Staubli VAL3: Piramide.pgx

program Piramide()
  local num j
  local num k
  local num i
  local num l
begin
  //Mueve el brazo para crear una pirámide en 3D.

  // Se desplaza a la posicion de espera
  pEspera=appro(pPieza,{0,0,-50,0,0,0})
  movej(pEspera,tVentosa,mNomSpeed)
  waitEndMove()

  //Ciclo
  while !bTermina
    if bStartPiramide
      // Bucle de plantas
      for i = 0 to nPlantas - 1
        // Bucle de filas
        for j = 0 to nPlantas - nNivel - 1
          // Bucle de piezas para fila central y superiores
          for k = 0 to nPlantas - nNivel - nFila - 1
            // Se espera la orden de pieza preparada para continuar
            sMensaje="pulse 'enter' para continuar"
            wait(bPiezaPreparada)
            bPiezaPreparada=false
            sMensaje=""

            pObjetivo = appro(pCentro,{nX,(nLPieza/2)*(nPlantas-nNivel-nFila-1)-nY,-nZ,0,0,0})
            call pick(pPieza,tVentosa,mNomSpeed,mVelApprox)
            call place(pObjetivo,tVentosa,mNomSpeed,mVelApprox)
            nY=nY+nLPieza
          endFor
          // Nueva fila, se reinician los valores de nY y aumenta nCont que calcula un nuevo valor para nX
          nY=0
          nCont=nCont+1
          //nX aumenta para hacer una fila inferior a continuación
          nX=nX+nWPieza*nCont
          //Aumenta nFila para disminuir nº de piezas por cada fila
          nFila=nFila+1
          // Se repite el bucle de piezas para hacer también las filas inferiores
          for l = 0 to nPlantas - nNivel - nFila - 1
            // Se espera la orden de pieza preparada para continuar
            sMensaje="pulse 'enter' para continuar"
            wait(bPiezaPreparada)
            bPiezaPreparada=false
            sMensaje=""

            pObjetivo = appro(pCentro,{nX,(nLPieza/2)*(nPlantas-nNivel-nFila-1)-nY,-nZ,0,0,0})
            call pick(pPieza,tVentosa,mNomSpeed,mVelApprox)
            call place(pObjetivo,tVentosa,mNomSpeed,mVelApprox)
            nY=nY+nLPieza
          endFor
          // Nueva fila, se reinician los valores de nY y aumenta nCont que calcula un nuevo valor para nX
          nY=0
          nCont=nCont+1
          //nX disminuye para hacer una fila superior a continuación
          nX=nX-nWPieza*nCont
        endFor
        //Nueva planta, se reinician los valores nX, nFila y nCont y aumentan nZ y nNivel
        nX=0
        nZ=nZ+12
        nFila=0
        nCont=0
        nNivel=nNivel+1
      endFor
      bStartPiramide=false
    endIf

    // Se le da paso a la siguiente tarea
    delay(0)
  endWhile
  bTermina=false

  // Se vuelve a la posicion de orgien
  movej(jHome,tVentosa,mNomSpeed)
  waitEndMove()

  bFin=true

end
